Fanuc KAREL source: kt00918.KL

PROGRAM KT00918
%STACKSIZE=65535
%PRIORITY=65535
%NOLOCKGROUP
VAR
S1 : STRING[80]
S2 : STRING[80]
OUT : INTEGER
BEGIN
S1='A'
S2='B'
S1='A'
S2='B'
-- UNRESOLVED_PC line 12 opcodes [27 22 2A 22 2A 76 23] marker_code=56
END KT00918
